Staubli VAL3: encodeJointData.pgx

public program encodeJointData(num& x_nStatus (dimensions=1), num& x_nOutputBuffer[] (dimensions=1), num& x_nBufferPos (dimensions=1), num& x_nJointData[] (dimensions=1))
  local num l_nDWordBytes[4]
  local num i
begin
  if x_nStatus<0
    return
  endIf
  x_nStatus=0
  for i=0 to size(x_nJointData)-1
    call encodeShareReal(x_nStatus,x_nOutputBuffer,x_nBufferPos,x_nJointData[i])
    if x_nStatus<0
      putln("Failed to encode joint data at index: "+toString("",x_nBufferPos)+" with "+toString("",x_nJointData[i]))
      return
    endIf
  endFor
end
